INTERFACE I_TaskCreator

METHOD create_future : I_Future
VAR_INPUT
	future_name :STRING; // Specify future name
END_VAR
END_METHOD

METHOD destroy_future : I_Future
VAR_INPUT
	future : I_Future; // Specify future instance whtat you want to delete.
END_VAR
END_METHOD

END_INTERFACE

(* stored: Version 1.1.0.1, ProductVersion 3.1.4026.17
   Itf I_TaskCreator: Id {5a160255-cfe3-43e1-811b-0ee8dbed2e75}
   Method create_future: Id {ea5b098b-00b2-478e-aedf-81f612d40841}
   Method destroy_future: Id {15f94faf-ca5d-40d1-a839-33168d7f650c} *)
